# B&R Automation Studio project brdkCert
Automation Studio 4.12.5.95 SP; technology packages: mapp 5.23.1, mappView 5.23.0

## Configuration Config1

CPU X20CP0484, AutomationRuntime H4.93, Build 4.1.2, Safety 0.0, Vc 

### Task classes (Cpu.sw)
```
Cyclic#1 (cycle 10000 us, tolerance 10000 us):
  ThirdParty <- SendThirdPartyToPanel.prg
Binaries: FWRules, mvLoader, TCData, udbdef, iomap, asfw, User, sysconf, arconfig, ashwd, Role, ashwac
Libraries: brdkCert, FileIO, runtime, standard, ArCert, astime, asieccon, arssl, AsIODiag, AsBrStr
```

### Hardware
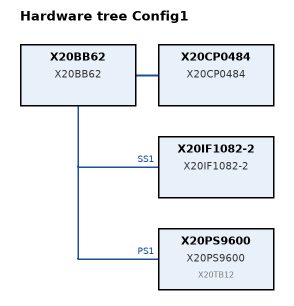
```
X20BB62 : X20BB62 v1.3.0.0
X20CP0484 : X20CP0484 v1.8.1.0  [SL -> X20BB62.SL1]
  Connector IF2:
    ActivateDevice = 1
    ActivateSnmp = 2
  ConfigurationID = brdkCert_Config1
  ConfigVersion = 1.0.1
  UserPartitionSize = 100
  EnableUsbRemoteInstall = 1
  EnableCfRemoteInstall = 1
  TimerDeviceType = SWIOTIMER
  Cyclic1Duration = 10000
  Cyclic1Tolerance = 10000
  Cyclic2Duration = 20000
  Cyclic2Tolerance = 20000
  Cyclic3Duration = 50000
  Cyclic3Tolerance = 50000
  Cyclic4Duration = 100000
  Cyclic4Tolerance = 100000
  Cyclic5Duration = 200000
  Cyclic5Tolerance = 200000
  Cyclic6Duration = 500000
  Cyclic6Tolerance = 500000
  Cyclic7Duration = 1000000
  Cyclic7Tolerance = 1000000
  Cyclic8Duration = 10000
  Cyclic8Tolerance = 30000000
  FileDevice1
  FileDeviceName1 = USER
  FileDevicePath1 = USER_PATH
  FtpUser1
  FtpUsername1 = admin
  FtpUserPassword1 = mdREweQc3UW/pA97MKi4oT9bNkw/h+8eCfsc7z3A7DE=
  FtpUserSalt1 = HOI4QVLF
  FTPAccessRight1 = 0
X20IF1082-2 : X20IF1082-2 v1.15.0.0  [SS -> X20BB62.SS1]
  Connector IF1:
    Operation = EthOnly
    ActivateANSL = 1
    ActivateSnmp = 2
X20PS9600 : X20PS9600 v1.6.1.0  [PS -> X20BB62.PS1; SS1 -> X20TB12.SS]
X20TB12 : X20TB12 v1.0.0.0
```

## Logical view

Binary libraries used (declarations not repeated): operator, runtime, astime, AsIecCon, FileIO, standard, ArCert, AsIODiag, AsBrStr

### Package Logical/Libraries - Global libraries

### Library Logical/Libraries/brdkCert (IEC) - Library to handle certificates
Depends on: FileIO, ArCert, AsBrStr

#### Types.typ - Exported data types
```iecst
TYPE
	brdk_cert_panel_type_typ :
		( (*Panel type.*)
		BRDK_CERT_NOT_IDENTIFIED := 0, (*Not identified.*)
		BRDK_CERT_T30 := 1, (*T30 panel.*)
		BRDK_CERT_T50 := 2, (*T50 panel.*)
		BRDK_CERT_T80 := 3, (*T80 panel.*)
		BRDK_CERT_FT50 := 4, (*FT50 panel.*)
		BRDK_CERT_MT50 := 5 (*MT50 panel.*)
		) := BRDK_CERT_NOT_IDENTIFIED;
END_TYPE
```

#### Constants.var - Exported constants
```iecst
VAR CONSTANT
	MAX_CERT_BUFFER_SIZE_IDX : UINT := 4999;
	MAX_CERT_SEND_IDX : UINT := 19;
END_VAR
```

#### brdkCert.fun - Exported functions and function blocks
```iecst
FUNCTION_BLOCK SendThirdPartyToPanel (*Will send a certificate from Third Party directry in AS to panel (ex. T80)*)
	VAR_INPUT
		Execute : BOOL;
		PanelEndpoint : STRING[16]; (*Endpoint to panel (IP)*)
		PanelType : brdk_cert_panel_type_typ;
		PanelPassword : STRING[10]; (*Password for usershare (configured in panel service menu)*)
		CertificateName : STRING[80]; (*'Example.cer" or "Example.crt"*)
		Simulated : BOOL;
	END_VAR
	VAR_OUTPUT
		Done : BOOL;
		Error : BOOL;
		BufferTooSmall : BOOL; (*Buffer too small for used certificate. Please increase "MAX_CERT_BUFFER_SIZE_IDX"*)
	END_VAR
	VAR
		state : USINT;
		ArCertExportThirdParty_0 : ArCertExportThirdParty;
		DevLink_0 : DevLink;
		DirCreate_0 : DirCreate;
		FileDelete_0 : FileDelete;
		FileCreate_0 : FileCreate;
		FileOpen_0 : FileOpen;
		FileWriteEx_0 : FileWriteEx;
		FileClose_0 : FileClose;
		DevUnlink_0 : DevUnlink;
		handle : UDINT;
		cifsParam : STRING[120]; (*Parameters to connect to panel usershare*)
		certBuffer : ARRAY[0..MAX_CERT_BUFFER_SIZE_IDX] OF USINT; (*Increase if certificate size exceeds "MAX_CERT_BUFFER_SIZE"*)
		filePath : STRING[50];
		fileIdent : UDINT;
		fileDeviceName : STRING[10];
	END_VAR
END_FUNCTION_BLOCK

FUNCTION_BLOCK SendListThirdPartyToPanel (*Will send a certificate from Third Party directry in AS to panel (ex. T80)*)
	VAR_INPUT
		Execute : BOOL;
		PanelEndpoint : STRING[16]; (*Endpoint to panel (IP)*)
		PanelType : brdk_cert_panel_type_typ;
		PanelPassword : STRING[10]; (*Password for usershare (configured in panel service menu)*)
		CertificateName : ARRAY[0..MAX_CERT_SEND_IDX] OF STRING[80]; (*'Example.cer" or "Example.crt"*)
		Simulated : BOOL;
	END_VAR
	VAR_OUTPUT
		Done : BOOL;
		Error : BOOL;
		BufferTooSmall : BOOL; (*Buffer too small for used certificate. Please increase "MAX_CERT_BUFFER_SIZE_IDX"*)
	END_VAR
	VAR
		state : USINT;
		ArCertExportThirdParty_0 : ArCertExportThirdParty;
		DevLink_0 : DevLink;
		DirCreate_0 : DirCreate;
		FileDelete_0 : FileDelete;
		FileCreate_0 : FileCreate;
		FileOpen_0 : FileOpen;
		FileWriteEx_0 : FileWriteEx;
		FileClose_0 : FileClose;
		DevUnlink_0 : DevUnlink;
		handle : UDINT;
		cifsParam : STRING[120]; (*Parameters to connect to panel usershare*)
		certBuffer : ARRAY[0..MAX_CERT_BUFFER_SIZE_IDX] OF USINT; (*Increase if certificate size exceeds "MAX_CERT_BUFFER_SIZE"*)
		filePath : STRING[50];
		fileIdent : UDINT;
		fileDeviceName : STRING[10];
	END_VAR
END_FUNCTION_BLOCK
```

#### SendThirdPartyToPanel.st
```iecst
FUNCTION_BLOCK SendThirdPartyToPanel

	IF NOT Execute AND state > 0 THEN
		state := 222; // will reset everything and return to state 0
	END_IF

	CASE state OF

		0:
			IF Execute THEN
				brsmemset(ADR(certBuffer),0,SIZEOF(certBuffer));

				// Connect to panel usershare
				cifsParam := CONCAT('/SIP=',PanelEndpoint);
				cifsParam := CONCAT(cifsParam,' /PROTOCOL=cifs /SHARE=usershare /USER=');
				CASE PanelType OF
					BRDK_CERT_T30: 	cifsParam := CONCAT(cifsParam,'ppts30-user'); ;
					BRDK_CERT_T50:	cifsParam := CONCAT(cifsParam,'ppts50-user'); ;
					BRDK_CERT_T80: 	cifsParam := CONCAT(cifsParam,'ppt80-user'); ;
					BRDK_CERT_FT50: cifsParam := CONCAT(cifsParam,'pft50-user'); ;
					BRDK_CERT_MT50:	cifsParam := CONCAT(cifsParam,'pmt50-user'); ;
				END_CASE
				cifsParam := CONCAT(cifsParam,' /PASSWORD=');
				cifsParam := CONCAT(cifsParam,PanelPassword);

				IF Simulated THEN
					fileDeviceName := 'USER';			// Use existing 'USER' file device if simulated
					state := 20;
				ELSE
					fileDeviceName := 'PANELCERT';		// Create file device 'PANELCERT' to usershare if real hardware.
					state := 10;
				END_IF

			END_IF

		10:
			DevLink_0.enable := TRUE;
			DevLink_0.pDevice := ADR(fileDeviceName);
			DevLink_0.pParam := ADR(cifsParam);
			DevLink_0();

			IF DevLink_0.status = ERR_OK OR DevLink_0.status = fiERR_DEVICE_ALREADY_EXIST THEN
				handle := DevLink_0.handle;
				DevLink_0.enable := FALSE;
				DevLink_0();
				state := 20;
			ELSIF DevLink_0.status <> ERR_FUB_BUSY THEN
				state := 222;
			END_IF

		20:
			ArCertExportThirdParty_0.Execute := TRUE;
			ArCertExportThirdParty_0.Name := CertificateName;
			ArCertExportThirdParty_0.Data := ADR(certBuffer);
			ArCertExportThirdParty_0.DataSize := SIZEOF(certBuffer);
			ArCertExportThirdParty_0();

			IF ArCertExportThirdParty_0.Error THEN
				state := 222;
			ELSIF ArCertExportThirdParty_0.Done AND NOT ArCertExportThirdParty_0.Busy THEN
				ArCertExportThirdParty_0.Execute := FALSE;
				ArCertExportThirdParty_0();

				IF ArCertExportThirdParty_0.NeededDataSize > MAX_CERT_BUFFER_SIZE_IDX THEN
					// If certificate size is bigger than the buffer we can't store it.
					BufferTooSmall := TRUE;
					state := 222;
				ELSE
					state := 30;
				END_IF

			END_IF

		30:
			DirCreate_0.enable := TRUE;
			DirCreate_0.pDevice := ADR(fileDeviceName);
			DirCreate_0.pName := ADR('cert');
			DirCreate_0();

			IF DirCreate_0.status = ERR_OK OR DirCreate_0.status = fiERR_DIR_ALREADY_EXIST THEN
				DirCreate_0.enable := FALSE;
				DirCreate_0();
				filePath := CONCAT('cert\',CertificateName);
				state := 40;
			ELSIF DirCreate_0.status <> ERR_FUB_BUSY THEN
				state := 222;
			END_IF

		40:
			FileCreate_0.enable := TRUE;
			FileCreate_0.pDevice := ADR(fileDeviceName);
			FileCreate_0.pFile := ADR(filePath);
			FileCreate_0();

			IF FileCreate_0.status = ERR_OK THEN
				fileIdent := FileCreate_0.ident;
				FileCreate_0.enable := FALSE;
				FileCreate_0();
				state := 60;
			ELSIF FileCreate_0.status = fiERR_EXIST THEN
				// File already exist -> use FileOpen instead.
				FileCreate_0.enable := FALSE;
				FileCreate_0();
				state := 50;
			ELSIF FileCreate_0.status <> ERR_FUB_BUSY THEN
				state := 222;
			END_IF

		50:
			FileOpen_0.enable := TRUE;
			FileOpen_0.pDevice := ADR(fileDeviceName);
			FileOpen_0.pFile := ADR(filePath);
			FileOpen_0.mode := FILE_W;
			FileOpen_0();

			IF FileOpen_0.status = ERR_OK THEN
				fileIdent := FileOpen_0.ident;
				FileOpen_0.enable := FALSE;
				FileOpen_0();
				state := 60;
			ELSIF FileOpen_0.status <> ERR_FUB_BUSY THEN
				state := 222;
			END_IF

		60:
			FileWriteEx_0.enable := TRUE;
			FileWriteEx_0.ident := fileIdent;
			FileWriteEx_0.pSrc := ADR(certBuffer);
			FileWriteEx_0.len := ArCertExportThirdParty_0.NeededDataSize;
			FileWriteEx_0.option := fiTruncate; // Will truncate (remove) any existing bytes after "FileWriteEx_0.len"
			FileWriteEx_0();

			IF FileWriteEx_0.status = ERR_OK THEN
				FileWriteEx_0.enable := FALSE;
				FileWriteEx_0();
				state := 70;
			ELSIF FileWriteEx_0.status <> ERR_FUB_BUSY THEN
				state := 222;
			END_IF

		70:
			FileClose_0.enable := TRUE;
			FileClose_0.ident := fileIdent;
			FileClose_0();

			IF FileClose_0.status = ERR_OK THEN
				FileClose_0.enable := FALSE;
				FileClose_0();
				state := SEL(Simulated,80,90);
			ELSIF FileClose_0.status <> ERR_FUB_BUSY THEN
				state := 222;
			END_IF

		80:
			DevUnlink_0.enable := TRUE;
			DevUnlink_0.handle := handle;
			DevUnlink_0();

			IF DevUnlink_0.status = ERR_OK THEN
				DevUnlink_0.enable := FALSE;
				DevUnlink_0();
				state := 90;
			ELSIF DevUnlink_0.status <> ERR_FUB_BUSY THEN
				DevUnlink_0.enable := FALSE;
				DevUnlink_0();
				state := 90;
			END_IF

		90:

			Done := TRUE;

			IF NOT Execute THEN
				Done := FALSE;
				state := 0;
			END_IF

		222:

			Error := TRUE;

			IF NOT Execute THEN
				// Reset everything
				ArCertExportThirdParty_0.Execute := FALSE;
				ArCertExportThirdParty_0();
				DevLink_0.enable := FALSE;
				DevLink_0();
				DirCreate_0.enable := FALSE;
				DirCreate_0();
				FileDelete_0.enable := FALSE;
				FileDelete_0();
				FileCreate_0.enable := FALSE;
				FileCreate_0();
				FileOpen_0.enable := FALSE;
				FileOpen_0();
				FileWriteEx_0.enable := FALSE;
				FileWriteEx_0();
				FileClose_0.enable := FALSE;
				FileClose_0();
				DevUnlink_0.enable := FALSE;
				DevUnlink_0();

				BufferTooSmall := FALSE;
				Error := FALSE;
				Done := FALSE;
				state := 0;
			END_IF

	END_CASE

END_FUNCTION_BLOCK
```

#### SendListThirdPartyToPanel.st
```iecst
FUNCTION_BLOCK SendListThirdPartyToPanel

	IF NOT Execute AND state > 0 THEN
		state := 222; // will reset everything and return to state 0
	END_IF

	CASE state OF

		0:
			IF Execute THEN
				brsmemset(ADR(certBuffer),0,SIZEOF(certBuffer));

				// Connect to panel usershare
				cifsParam := CONCAT('/SIP=',PanelEndpoint);
				cifsParam := CONCAT(cifsParam,' /PROTOCOL=cifs /SHARE=usershare /USER=');
				CASE PanelType OF
					BRDK_CERT_T30: 	cifsParam := CONCAT(cifsParam,'ppts30-user'); ;
					BRDK_CERT_T50:	cifsParam := CONCAT(cifsParam,'ppts50-user'); ;
					BRDK_CERT_T80: 	cifsParam := CONCAT(cifsParam,'ppt80-user'); ;
					BRDK_CERT_FT50: cifsParam := CONCAT(cifsParam,'pft50-user'); ;
					BRDK_CERT_MT50:	cifsParam := CONCAT(cifsParam,'pmt50-user'); ;
				END_CASE
				cifsParam := CONCAT(cifsParam,' /PASSWORD=');
				cifsParam := CONCAT(cifsParam,PanelPassword);

				IF Simulated THEN
					fileDeviceName := 'USER';		// Use existing 'USER' file device if simulated
					state := 20;
				ELSE
					fileDeviceName := 'PANEL';		// Create file device 'PANEL' to usershare if real hardware.
					state := 10;
				END_IF

			END_IF

		10:
			DevLink_0.enable := TRUE;
			DevLink_0.pDevice := ADR(fileDeviceName);
			DevLink_0.pParam := ADR(cifsParam);
			DevLink_0();

			IF DevLink_0.status = ERR_OK OR DevLink_0.status = fiERR_DEVICE_ALREADY_EXIST THEN
				handle := DevLink_0.handle;
				DevLink_0.enable := FALSE;
				DevLink_0();
				state := 20;
			ELSIF DevLink_0.status <> ERR_FUB_BUSY THEN
				state := 222;
			END_IF

		20:
			ArCertExportThirdParty_0.Execute := TRUE;
			ArCertExportThirdParty_0.Name := CertificateName;
			ArCertExportThirdParty_0.Data := ADR(certBuffer);
			ArCertExportThirdParty_0.DataSize := SIZEOF(certBuffer);
			ArCertExportThirdParty_0();

			IF ArCertExportThirdParty_0.Error THEN
				state := 222;
			ELSIF ArCertExportThirdParty_0.Done AND NOT ArCertExportThirdParty_0.Busy THEN
				ArCertExportThirdParty_0.Execute := FALSE;
				ArCertExportThirdParty_0();

				IF ArCertExportThirdParty_0.NeededDataSize > MAX_CERT_BUFFER_SIZE_IDX THEN
					// If certificate size is bigger than the buffer we can't store it.
					BufferTooSmall := TRUE;
					state := 222;
				ELSE
					state := 30;
				END_IF

			END_IF

		30:
			DirCreate_0.enable := TRUE;
			DirCreate_0.pDevice := ADR(fileDeviceName);
			DirCreate_0.pName := ADR('cert');
			DirCreate_0();

			IF DirCreate_0.status = ERR_OK OR DirCreate_0.status = fiERR_DIR_ALREADY_EXIST THEN
				DirCreate_0.enable := FALSE;
				DirCreate_0();
				filePath := CONCAT('cert\',CertificateName);
				state := 40;
			ELSIF DirCreate_0.status <> ERR_FUB_BUSY THEN
				state := 222;
			END_IF

		40:
			FileCreate_0.enable := TRUE;
			FileCreate_0.pDevice := ADR(fileDeviceName);
			FileCreate_0.pFile := ADR(filePath);
			FileCreate_0();

			IF FileCreate_0.status = ERR_OK THEN
				fileIdent := FileCreate_0.ident;
				FileCreate_0.enable := FALSE;
				FileCreate_0();
				state := 60;
			ELSIF FileCreate_0.status = fiERR_EXIST THEN
				// File already exist -> use FileOpen instead.
				FileCreate_0.enable := FALSE;
				FileCreate_0();
				state := 50;
			ELSIF FileCreate_0.status <> ERR_FUB_BUSY THEN
				state := 222;
			END_IF

		50:
			FileOpen_0.enable := TRUE;
			FileOpen_0.pDevice := ADR(fileDeviceName);
			FileOpen_0.pFile := ADR(filePath);
			FileOpen_0.mode := FILE_W;
			FileOpen_0();

			IF FileOpen_0.status = ERR_OK THEN
				fileIdent := FileOpen_0.ident;
				FileOpen_0.enable := FALSE;
				FileOpen_0();
				state := 60;
			ELSIF FileOpen_0.status <> ERR_FUB_BUSY THEN
				state := 222;
			END_IF

		60:
			FileWriteEx_0.enable := TRUE;
			FileWriteEx_0.ident := fileIdent;
			FileWriteEx_0.pSrc := ADR(certBuffer);
			FileWriteEx_0.len := ArCertExportThirdParty_0.NeededDataSize;
			FileWriteEx_0.option := fiTruncate; // Will truncate (remove) any existing bytes after "FileWriteEx_0.len"
			FileWriteEx_0();

			IF FileWriteEx_0.status = ERR_OK THEN
				FileWriteEx_0.enable := FALSE;
				FileWriteEx_0();
				state := 70;
			ELSIF FileWriteEx_0.status <> ERR_FUB_BUSY THEN
				state := 222;
			END_IF

		70:
			FileClose_0.enable := TRUE;
			FileClose_0.ident := fileIdent;
			FileClose_0();

			IF FileClose_0.status = ERR_OK THEN
				FileClose_0.enable := FALSE;
				FileClose_0();
				state := SEL(Simulated,80,90);
			ELSIF FileClose_0.status <> ERR_FUB_BUSY THEN
				state := 222;
			END_IF

		80:
			DevUnlink_0.enable := TRUE;
			DevUnlink_0.handle := handle;
			DevUnlink_0();

			IF DevUnlink_0.status = ERR_OK THEN
				DevUnlink_0.enable := FALSE;
				DevUnlink_0();
				state := 90;
			ELSIF DevUnlink_0.status <> ERR_FUB_BUSY THEN
				state := 222;
			END_IF

		90:

			Done := TRUE;

			IF NOT Execute THEN
				Done := FALSE;
				state := 0;
			END_IF

		222:

			Error := TRUE;

			IF NOT Execute THEN
				// Reset everything
				ArCertExportThirdParty_0.Execute := FALSE;
				ArCertExportThirdParty_0();
				DevLink_0.enable := FALSE;
				DevLink_0();
				DirCreate_0.enable := FALSE;
				DirCreate_0();
				FileDelete_0.enable := FALSE;
				FileDelete_0();
				FileCreate_0.enable := FALSE;
				FileCreate_0();
				FileOpen_0.enable := FALSE;
				FileOpen_0();
				FileWriteEx_0.enable := FALSE;
				FileWriteEx_0();
				FileClose_0.enable := FALSE;
				FileClose_0();
				DevUnlink_0.enable := FALSE;
				DevUnlink_0();

				BufferTooSmall := FALSE;
				Error := FALSE;
				Done := FALSE;
				state := 0;
			END_IF

	END_CASE

END_FUNCTION_BLOCK
```

### Program Logical/SendThirdPartyToPanel (IEC)

#### Main.st
```iecst
PROGRAM _INIT

	SendThirdPartyToPanel_0.PanelEndpoint := '192.168.30.222';
	SendThirdPartyToPanel_0.PanelType := BRDK_CERT_FT50;
	SendThirdPartyToPanel_0.PanelPassword := '1234';
	SendThirdPartyToPanel_0.CertificateName := 'e6.cer';

	SendThirdPartyToPanel_0.Simulated := DiagCpuIsARsim();
END_PROGRAM

PROGRAM _CYCLIC

	SendThirdPartyToPanel_0();

END_PROGRAM

PROGRAM _EXIT

END_PROGRAM
```

### Program Logical/SendListThirdPartyToPanel (IEC)

#### Variables.var
```iecst
VAR
	SendListThirdPartyToPanel_0 : SendListThirdPartyToPanel;
END_VAR
```

#### Main.st
```iecst
PROGRAM _INIT

	SendListThirdPartyToPanel_0.PanelEndpoint := '192.168.30.222';
	SendListThirdPartyToPanel_0.PanelType := BRDK_CERT_FT50;
	SendListThirdPartyToPanel_0.PanelPassword := '1234';
	SendListThirdPartyToPanel_0.CertificateName[0] := 'e6.cer';
	SendListThirdPartyToPanel_0.CertificateName[1] := 'r11.cer';
	SendListThirdPartyToPanel_0.CertificateName[2] := 'r10.cer';
	SendListThirdPartyToPanel_0.CertificateName[3] := 'isrg-root-x2-cross-signed.cer';
	SendListThirdPartyToPanel_0.CertificateName[4] := 'isrg-root-x1-cross-signed.cer';
	SendListThirdPartyToPanel_0.CertificateName[5] := 'e5.cer';
	SendListThirdPartyToPanel_0.CertificateName[6] := '1282303295.crt';

	SendListThirdPartyToPanel_0.Simulated := DiagCpuIsARsim();
END_PROGRAM

PROGRAM _CYCLIC

	SendListThirdPartyToPanel_0();

END_PROGRAM

PROGRAM _EXIT

END_PROGRAM
```

### Variables.var
```iecst
VAR
	SendThirdPartyToPanel_0 : SendThirdPartyToPanel;
END_VAR
```

Listed in the project but not available here: Logical/Global.typ, Logical/Global.var
